{attribute 'conditionalshow'}
TYPE PositionExtremaDesc :
STRUCT
  Minimum, Maximum : LREAL; // The extreme position
  Tmin, Tmax : LREAL;  // Time when the positions are reached
END_STRUCT
END_TYPE

(* stored: Version 1.1.0.1
   DUT PositionExtremaDesc: Id {b615dcba-8544-436f-9a57-30985945064e} *)
